(* IEC 61131-3 sources: test/Class/_SyncTimeHMI, 1 file *)

(* ---- _SyncTimeHMI.st ---- *)
(*!
<Class
	Name               = "_SyncTimeHMI"
	Revision           = "2.2"
	RealtimeTask       = "false"
	CyclicTask         = "false"
	BackgroundTask     = "true"
	DefBackground      = "100 ms"
	Sigmatek           = "true"
	OSInterface        = "false"
	HighPriority       = "false"
	Automatic          = "false"
	UpdateMode         = "Prescan"
	SharedCommandTable = "true"
	Objectsize         = "(540,180)"
	Comment            = "class reads date and time from two clients (within the adjusted zycletime)&#13;&#10;and writes these values to the servers">
	<Channels>
		<Server Name="sSyncDate" Visualized="true" Initialize="false" WriteProtected="false" Retentive="false" Comment="server for sync date - also input is possible"/>
		<Server Name="sSyncTime" Visualized="true" Initialize="false" WriteProtected="false" Retentive="false" Comment="server for sync time - also input is possible"/>
		<Server Name="SyncFromMc" Visualized="false" Initialize="true" DefValue="0" WriteProtected="false" Retentive="false" Comment="0 ... synchronisation is done from HMI to MC&#13;&#10;1 ... synchronisation is done from MC to HMI (needed when there is no RTC on the HMI"/>
		<Server Name="SyncInterval" Visualized="true" Initialize="true" DefValue="20sec" WriteProtected="false" Retentive="false" Comment="[ms] the time will be checked after this time has elapsed"/>
		<Client Name="ActDate" Required="true" Internal="false" Comment="actual date"/>
		<Client Name="ActTime" Required="true" Internal="false" Comment="actual time"/>
		<Client Name="Online" Required="false" Internal="false" Comment="connect this client to ensure, that the connected source can provide the correct&#13;&#10;values, this is important when the server &quot;SyncFromMc&quot; is set to 1"/>
		<Client Name="SetDate" Required="false" Internal="false" Comment="destination date (e.g. for Machine Control)"/>
		<Client Name="SetTime" Required="false" Internal="false" Comment="destination time (e.g. for Machine Control)"/>
	</Channels>
	<Dependencies>
		<Files>
			<File Path=".\Class\_SyncTimeHMI\_SyncTimeHMI_de.pdf"/>
			<File Path=".\Class\_SyncTimeHMI\_SyncTimeHMI_en.pdf"/>
		</Files>
	</Dependencies>
	<RevDoku>
		<Owner Company="Sigmatek" Author="FurLuk"/>
		<Dokumentation Revision="2.2" Date="2021-08-11" Author="HasHan" Company="Sigmatek" Description="Improvement: implementation of the online-client&#13;&#10;Improvement: implementation of the SyncInterval-server"/>
		<Dokumentation Revision="2.1" Date="2019-07-11" Author="FurLuk" Company="Sigmatek" Description="added server SyncFromMc in order to be able to synchronise time form the MachineControll to the HMI"/>
		<Dokumentation Revision="2.0" Date="2018-02-07" Author="KaiAnd" Company="Sigmatek" Description="Implemented functionality to take over date &amp; time of inputs on server vars&#13;&#10;--&gt; server for date &amp; time now have write() mwthods for inputs&#13;&#10;--&gt; new destination clients SetDate and SetTime (optional)"/>
		<Dokumentation Revision="1.1" Date="2016-10-10" Author="HubChr" Company="Sigmatek" Description="Added documentation pdfs."/>
		<Dokumentation Revision="1.0" Date="2015-11-11" Author="hötant" Company="Sigmatek" Description="creation of class"/>
	</RevDoku>
</Class>
*)
_SyncTimeHMI : CLASS
  //Servers:
	sSyncDate 	: SvrChCmd_DATE_LSL;
	sSyncTime 	: SvrCh_TIME_LSL;
	SyncFromMc 	: SvrCh_DINT;
	SyncInterval 	: SvrCh_UDINT;
  //Clients:
	ActDate 	: CltCh_HDINT;
	ActTime 	: CltCh_HDINT;
	SetDate 	: CltCh_HDINT;
	SetTime 	: CltCh_HDINT;
	Online 	: CltCh_DINT;
  //Variables:
		IsCon_SetDate 	: DINT;			//! <Variable Comment="&quot;Is Connected&quot; flag ..." Name="IsCon_SetDate"/>
		IsCon_SetTime 	: DINT;			//! <Variable Comment="&quot;Is Connected&quot; flag ..." Name="IsCon_SetTime"/>
		TimeStampSync 	: UDINT;
		IsCon_Online 	: DINT;			//! <Variable Comment="&quot;Is Connected&quot; flag ..." Name="IsCon_Online"/>
  //Functions:

	FUNCTION VIRTUAL GLOBAL Init;

	FUNCTION VIRTUAL GLOBAL Background
		VAR_INPUT
			EAX 	: UDINT;
		END_VAR
		VAR_OUTPUT
			state (EAX) 	: UDINT;
		END_VAR;

	FUNCTION VIRTUAL GLOBAL sSyncDate::Read
		VAR_OUTPUT
			output (EAX) 	: DATE_LSL;
		END_VAR;

	FUNCTION VIRTUAL GLOBAL sSyncDate::Write
		VAR_INPUT
			input (EAX) 	: DATE_LSL;
		END_VAR
		VAR_OUTPUT
			result (EAX) 	: DATE_LSL;
		END_VAR;

	FUNCTION VIRTUAL GLOBAL sSyncTime::Read
		VAR_OUTPUT
			output (EAX) 	: TIME_LSL;
		END_VAR;

	FUNCTION VIRTUAL GLOBAL sSyncTime::Write
		VAR_INPUT
			input (EAX) 	: TIME_LSL;
		END_VAR
		VAR_OUTPUT
			result (EAX) 	: TIME_LSL;
		END_VAR;
  //Tables:
	FUNCTION @STD
		VAR_OUTPUT
			ret_code	: CONFSTATES;
		END_VAR;
	FUNCTION GLOBAL TAB @CT_;
END_CLASS;

FUNCTION VIRTUAL GLOBAL _SyncTimeHMI::Init

  if (_FirstScan) then

    IsCon_SetDate := IsCon_SetTime := IsCon_Online := 0;
    if (IsClientConnected(#SetDate)) then IsCon_SetDate := 1; end_if;
    if (IsClientConnected(#SetTime)) then IsCon_SetTime := 1; end_if;
    if (IsClientConnected(#Online))  then IsCon_Online  := 1; end_if;

  end_if;

END_FUNCTION

FUNCTION VIRTUAL GLOBAL _SyncTimeHMI::Background
	VAR_INPUT
		EAX 	: UDINT;
	END_VAR
	VAR_OUTPUT
		state (EAX) 	: UDINT;
	END_VAR

	state := READY;

  ActDate := ActDate.Read();
  ActTime := ActTime.Read();

  //-------------------------------------------------------------------------------------------------------------------
  if (SyncFromMc = 0) then //synchronise time from HMI to MC

    if ((ops.tAbsolute - TimeStampSync) >= SyncInterval) then
      TimeStampSync := ops.tAbsolute;

      if (IsCon_SetDate = TRUE) then
        SetDate := ActDate;
        SetDate.Write(ActDate);
      end_if;

      if (IsCon_SetTime = TRUE) then
        SetTime := ActTime;
        SetTime.Write(ActTime);
      end_if;

    end_if;

  //-------------------------------------------------------------------------------------------------------------------
  elsif (SyncFromMc = 1) then //synchronise time from MC to HMI

    if ((ops.tAbsolute - TimeStampSync) >= SyncInterval) then
      TimeStampSync := ops.tAbsolute;

      if (IsCon_Online = 1) & (Online.Read() = 0) then //is the Online-client connected?
        return; //the connection is not established yet, no valid data will be available at SetDate and SetTime
      end_if;

      if (IsCon_SetDate = TRUE) then
        SetDate := SetDate.Read();
        ActDate.Write(SetDate);
        ActDate := SetDate;
      end_if;

      if (IsCon_SetTime = TRUE) then
        SetTime := SetTime.Read();
        ActTime.Write(SetTime);
        ActTime := SetTime;
      end_if;

    end_if;

  end_if;

END_FUNCTION

FUNCTION VIRTUAL GLOBAL _SyncTimeHMI::sSyncDate::Read
	VAR_OUTPUT
		output (EAX) 	: DATE_LSL;
	END_VAR

 output := sSyncDate := ActDate := ActDate.Read();

END_FUNCTION

FUNCTION VIRTUAL GLOBAL _SyncTimeHMI::sSyncTime::Read
	VAR_OUTPUT
		output (EAX) 	: TIME_LSL;
	END_VAR

	output := sSyncTime := ActTime := ActTime.Read();

END_FUNCTION

FUNCTION VIRTUAL GLOBAL _SyncTimeHMI::sSyncDate::Write
	VAR_INPUT
		input (EAX) 	: DATE_LSL;
	END_VAR
	VAR_OUTPUT
		result (EAX) 	: DATE_LSL;
	END_VAR

	sSyncDate := input;
	result := sSyncDate;

  // write input date to destination
  ActDate := sSyncDate;
  ActDate.Write(sSyncDate);

  if (IsCon_SetDate = TRUE) then
    SetDate := sSyncDate;
    SetDate.Write(sSyncDate);
  end_if;

END_FUNCTION

FUNCTION VIRTUAL GLOBAL _SyncTimeHMI::sSyncTime::Write
	VAR_INPUT
		input (EAX) 	: TIME_LSL;
	END_VAR
	VAR_OUTPUT
		result (EAX) 	: TIME_LSL;
	END_VAR

	sSyncTime := input;
	result := sSyncTime;

  // write input time to destination
  ActTime := sSyncTime;
  ActTime.Write(sSyncTime);

  if (IsCon_SetTime = TRUE) then
    SetTime := sSyncTime;
    SetTime.Write(sSyncTime);
  end_if;

END_FUNCTION
